FUNCTION StringEndsWith : BOOL
VAR_INPUT
	text : T_MaxString;
	endsWithString : T_MaxString;
END_VAR
VAR
	textLength : DINT;
	length : DINT;
END_VAR

textLength := LEN(text);
length := LEN(endsWithString);

IF (textLength < length) THEN
	RETURN;
END_IF

StringEndsWith := MEMCMP(pBuf1 := ADR(text) + TO_DWORD(textLength - length), pBuf2 := ADR(endsWithString), n := TO_UDINT(length)) = 0;

END_FUNCTION

(* stored: Version 1.1.0.1
   POU StringEndsWith: Id {16faa171-6f34-01d0-1d79-268489938df3}, SpecialFunc None *)
